// TwinCAT 3 PLC project PLC1
// ProgramVersion: 3.1.4023.0
// libraries:
//   Tc2_Utilities, * (Beckhoff Automation GmbH)
//   CmpBitmapPool, * (System)
//   Tc2_ControllerToolbox, * (Beckhoff Automation GmbH)
//   Tc2_MC2, * (Beckhoff Automation GmbH)
//   Tc2_NC, * (Beckhoff Automation GmbH)
//   Tc2_Standard, * (Beckhoff Automation GmbH)
//   Tc2_System, * (Beckhoff Automation GmbH)
//   Tc3_IoLink, * (Beckhoff Automation GmbH)
//   Tc3_Module, * (Beckhoff Automation GmbH)
//   VisuDialogs, * (System)
//   VisuSymbols,3.5.10.0,System
// project tree:
//   DUTs/ Figure.TcDUT, Mode.TcDUT
//   DUTs/CyltronicCom/ CyltronicMotionMode.TcDUT, CyltronicProcessDataInActual.TcDUT, CyltronicProcessDataInBytes.TcDUT, CyltronicProcessDataIn.TcDUT, CyltronicProcessDataOut.TcDUT, CyltronicProcessDataOutActual.TcDUT, CyltronicProcessDataOutBytes.TcDUT, CyltronicState.TcDUT
//   / GlobalTextList.TcGTLO, ImagePool.TcIPO (not stored), PLC_TASK.TcTTO, VISU_TASK.TcTTO
//   GVLs/ Config.TcGVL, GVL.TcGVL
//   POUs/ CONTROLLER.TcPOU, FBCylTronicCylinder.TcPOU, FB_FigureGenerator.TcPOU, FB_FigurePlayer.TcPOU, FB_BallTrack.TcPOU, FB_ReglerParam.TcPOU, MAIN.TcPOU, Touchpanel.TcPOU, TOUCH_SCALE.TcPOU, xy_RST_Transformation_dynamisch.TcPOU
//   POUs/Regelungstechnik/ DT1.TcPOU, eFiltertyp.TcDUT, eReglertyp.TcDUT, eSignalform.TcDUT, FB_Totband.TcPOU, Integrator.TcPOU, Logger_RET.TcPOU, P.TcPOU, PT1.TcPOU, PT2.TcPOU, PT2s.TcPOU, PTt.TcPOU, Rauschen.TcPOU, Regler.TcPOU, RET_COMMON.TcPOU, Signalgenerator.TcPOU, Strecke.TcPOU
//   POUs/Regelungstechnik/visu/ RET_VISU_DT1.TcVIS, RET_VISU_Integrator.TcVIS, RET_VISU_Kennlinie.TcVIS, RET_VISU_P.TcVIS, RET_VISU_PT1.TcVIS, RET_VISU_PT2.TcVIS, RET_VISU_PT2s.TcVIS, RET_VISU_PTt.TcVIS, RET_VISU_Regler.TcVIS, RET_VISU_Signalgenerator.TcVIS, RET_VISU_Strecke.TcVIS, TextListForCombobox_eReglertyp.TcTLO, TextListForCombobox_eSignalform.TcTLO, VISU_HELPER_Combobox_eReglertyp.TcVIS, VISU_HELPER_Combobox_eSignalform.TcVIS
//   VISUs/ Achse_R.TcVIS, Achse_S.TcVIS, Achse_T.TcVIS, FigureGeneratorDisplay.TcVIS, Home.TcVIS, FigureGenerator1.TcVIS, Debug.TcVIS, InputNumSlider_Corner.TcVIS, InputNumSlider_Radius.TcVIS, InputNumSlider_Angle.TcVIS, InputNumSlider_Time.TcVIS, Mainvisu.TcVIS, Polygon.TcVIS, FigurePlayer.TcVIS, FigureGenerator.TcVIS, FigurePlayerDisplay.TcVIS, Polygon_1.TcVIS, VisualizationManager.TcVMO (not stored), Visu_Achse.TcVIS
// real-time tasks:
//   TASK PLC_TASK: cycle T#1ms, priority 1, ADS port 350
//   TASK VISU_TASK: cycle T#200000us, priority 12, ADS port 351
// I/O:
//   DEVICE Device 2 (EtherCAT), AmsNetId 192.168.0.33.3.1
//     Klemme 1 (EK1200) [EK1200-5000 EtherCAT Netzteil (2A E-Bus)]
//       Klemme 2 (EL6224) [EL6224 (IO Link Master)]
//       Klemme 3 (EL1859) [EL1859 8K. Dig. Eingang 24V, 3ms, 8K. Dig. Ausgang 24V, 0.5A]
//       Klemme 4 (EK1110) [EK1110 EtherCAT-Verlängerung]
//     Box 14 (ABBTS Ball and Plate) [ABBTS Ball and Plate]
// variable links:
//   PLC1/PLC1 Instance <-> Device 2 (EtherCAT)/Box 14 (ABBTS Ball and Plate)
//     PLC_TASK Inputs/Touchpanel.bContactAvailable <-> Inputs/byContactAvailable
//     PLC_TASK Inputs/Touchpanel.iXadc <-> Inputs/iXraw
//     PLC_TASK Inputs/Touchpanel.iYadc <-> Inputs/iYraw
//     PLC_TASK Inputs/Touchpanel.iZadc <-> Inputs/iZraw
//     PLC_TASK Inputs/Touchpanel.rXadc <-> Inputs/rX
//     PLC_TASK Inputs/Touchpanel.rYadc <-> Inputs/rY
//     PLC_TASK Inputs/Touchpanel.rZadc <-> Inputs/rZ
//     PLC_TASK Outputs/Touchpanel.iStep <-> Outputs/iStep
//     PLC_TASK Outputs/Touchpanel.rQ_Kalman <-> Outputs/rQ_Kalman
//     PLC_TASK Outputs/Touchpanel.rR_Kalman <-> Outputs/rR_Kalman
//   PLC1/PLC1 Instance <-> Device 2 (EtherCAT)/Term 1 (EK1200)/Term 2 (EL6224)
//     PLC_TASK Inputs/MAIN.Axis_R.DataIn/CyltronicDataInByte/Byte0 <-> IO-Link Port1_in/SubIndex 001[0]
//     PLC_TASK Inputs/MAIN.Axis_R.DataIn/CyltronicDataInByte/Byte1 <-> IO-Link Port1_in/SubIndex 001[1]
//     PLC_TASK Inputs/MAIN.Axis_R.DataIn/CyltronicDataInByte/Byte10 <-> IO-Link Port1_in/SubIndex 001[10]
//     PLC_TASK Inputs/MAIN.Axis_R.DataIn/CyltronicDataInByte/Byte11 <-> IO-Link Port1_in/SubIndex 001[11]
//     PLC_TASK Inputs/MAIN.Axis_R.DataIn/CyltronicDataInByte/Byte12 <-> IO-Link Port1_in/SubIndex 001[12]
//     PLC_TASK Inputs/MAIN.Axis_R.DataIn/CyltronicDataInByte/Byte13 <-> IO-Link Port1_in/SubIndex 001[13]
//     PLC_TASK Inputs/MAIN.Axis_R.DataIn/CyltronicDataInByte/Byte2 <-> IO-Link Port1_in/SubIndex 001[2]
//     PLC_TASK Inputs/MAIN.Axis_R.DataIn/CyltronicDataInByte/Byte3 <-> IO-Link Port1_in/SubIndex 001[3]
//     PLC_TASK Inputs/MAIN.Axis_R.DataIn/CyltronicDataInByte/Byte4 <-> IO-Link Port1_in/SubIndex 001[4]
//     PLC_TASK Inputs/MAIN.Axis_R.DataIn/CyltronicDataInByte/Byte5 <-> IO-Link Port1_in/SubIndex 001[5]
//     PLC_TASK Inputs/MAIN.Axis_R.DataIn/CyltronicDataInByte/Byte6 <-> IO-Link Port1_in/SubIndex 001[6]
//     PLC_TASK Inputs/MAIN.Axis_R.DataIn/CyltronicDataInByte/Byte7 <-> IO-Link Port1_in/SubIndex 001[7]
//     PLC_TASK Inputs/MAIN.Axis_R.DataIn/CyltronicDataInByte/Byte8 <-> IO-Link Port1_in/SubIndex 001[8]
//     PLC_TASK Inputs/MAIN.Axis_R.DataIn/CyltronicDataInByte/Byte9 <-> IO-Link Port1_in/SubIndex 001[9]
//     PLC_TASK Inputs/MAIN.Axis_S.DataIn/CyltronicDataInByte/Byte0 <-> IO-Link Port2_in/SubIndex 001[0]
//     PLC_TASK Inputs/MAIN.Axis_S.DataIn/CyltronicDataInByte/Byte1 <-> IO-Link Port2_in/SubIndex 001[1]
//     PLC_TASK Inputs/MAIN.Axis_S.DataIn/CyltronicDataInByte/Byte10 <-> IO-Link Port2_in/SubIndex 001[10]
//     PLC_TASK Inputs/MAIN.Axis_S.DataIn/CyltronicDataInByte/Byte11 <-> IO-Link Port2_in/SubIndex 001[11]
//     PLC_TASK Inputs/MAIN.Axis_S.DataIn/CyltronicDataInByte/Byte12 <-> IO-Link Port2_in/SubIndex 001[12]
//     PLC_TASK Inputs/MAIN.Axis_S.DataIn/CyltronicDataInByte/Byte13 <-> IO-Link Port2_in/SubIndex 001[13]
//     PLC_TASK Inputs/MAIN.Axis_S.DataIn/CyltronicDataInByte/Byte2 <-> IO-Link Port2_in/SubIndex 001[2]
//     PLC_TASK Inputs/MAIN.Axis_S.DataIn/CyltronicDataInByte/Byte3 <-> IO-Link Port2_in/SubIndex 001[3]
//     PLC_TASK Inputs/MAIN.Axis_S.DataIn/CyltronicDataInByte/Byte4 <-> IO-Link Port2_in/SubIndex 001[4]
//     PLC_TASK Inputs/MAIN.Axis_S.DataIn/CyltronicDataInByte/Byte5 <-> IO-Link Port2_in/SubIndex 001[5]
//     PLC_TASK Inputs/MAIN.Axis_S.DataIn/CyltronicDataInByte/Byte6 <-> IO-Link Port2_in/SubIndex 001[6]
//     PLC_TASK Inputs/MAIN.Axis_S.DataIn/CyltronicDataInByte/Byte7 <-> IO-Link Port2_in/SubIndex 001[7]
//     PLC_TASK Inputs/MAIN.Axis_S.DataIn/CyltronicDataInByte/Byte8 <-> IO-Link Port2_in/SubIndex 001[8]
//     PLC_TASK Inputs/MAIN.Axis_S.DataIn/CyltronicDataInByte/Byte9 <-> IO-Link Port2_in/SubIndex 001[9]
//     PLC_TASK Inputs/MAIN.Axis_T.DataIn/CyltronicDataInByte/Byte0 <-> IO-Link Port3_in/SubIndex 001[0]
//     PLC_TASK Inputs/MAIN.Axis_T.DataIn/CyltronicDataInByte/Byte1 <-> IO-Link Port3_in/SubIndex 001[1]
//     PLC_TASK Inputs/MAIN.Axis_T.DataIn/CyltronicDataInByte/Byte10 <-> IO-Link Port3_in/SubIndex 001[10]
//     PLC_TASK Inputs/MAIN.Axis_T.DataIn/CyltronicDataInByte/Byte11 <-> IO-Link Port3_in/SubIndex 001[11]
//     PLC_TASK Inputs/MAIN.Axis_T.DataIn/CyltronicDataInByte/Byte12 <-> IO-Link Port3_in/SubIndex 001[12]
//     PLC_TASK Inputs/MAIN.Axis_T.DataIn/CyltronicDataInByte/Byte13 <-> IO-Link Port3_in/SubIndex 001[13]
//     PLC_TASK Inputs/MAIN.Axis_T.DataIn/CyltronicDataInByte/Byte2 <-> IO-Link Port3_in/SubIndex 001[2]
//     PLC_TASK Inputs/MAIN.Axis_T.DataIn/CyltronicDataInByte/Byte3 <-> IO-Link Port3_in/SubIndex 001[3]
//     PLC_TASK Inputs/MAIN.Axis_T.DataIn/CyltronicDataInByte/Byte4 <-> IO-Link Port3_in/SubIndex 001[4]
//     PLC_TASK Inputs/MAIN.Axis_T.DataIn/CyltronicDataInByte/Byte5 <-> IO-Link Port3_in/SubIndex 001[5]
//     PLC_TASK Inputs/MAIN.Axis_T.DataIn/CyltronicDataInByte/Byte6 <-> IO-Link Port3_in/SubIndex 001[6]
//     PLC_TASK Inputs/MAIN.Axis_T.DataIn/CyltronicDataInByte/Byte7 <-> IO-Link Port3_in/SubIndex 001[7]
//     PLC_TASK Inputs/MAIN.Axis_T.DataIn/CyltronicDataInByte/Byte8 <-> IO-Link Port3_in/SubIndex 001[8]
//     PLC_TASK Inputs/MAIN.Axis_T.DataIn/CyltronicDataInByte/Byte9 <-> IO-Link Port3_in/SubIndex 001[9]
//     PLC_TASK Outputs/MAIN.Axis_R.DataOut/CyltronicDataOutByte/Byte0 <-> IO-Link Port1_out/SubIndex 001[0]
//     PLC_TASK Outputs/MAIN.Axis_R.DataOut/CyltronicDataOutByte/Byte1 <-> IO-Link Port1_out/SubIndex 001[1]
//     PLC_TASK Outputs/MAIN.Axis_R.DataOut/CyltronicDataOutByte/Byte2 <-> IO-Link Port1_out/SubIndex 001[2]
//     PLC_TASK Outputs/MAIN.Axis_R.DataOut/CyltronicDataOutByte/Byte3 <-> IO-Link Port1_out/SubIndex 001[3]
//     PLC_TASK Outputs/MAIN.Axis_R.DataOut/CyltronicDataOutByte/Byte4 <-> IO-Link Port1_out/SubIndex 001[4]
//     PLC_TASK Outputs/MAIN.Axis_R.DataOut/CyltronicDataOutByte/Byte5 <-> IO-Link Port1_out/SubIndex 001[5]
//     PLC_TASK Outputs/MAIN.Axis_R.DataOut/CyltronicDataOutByte/Byte6 <-> IO-Link Port1_out/SubIndex 001[6]
//     PLC_TASK Outputs/MAIN.Axis_R.DataOut/CyltronicDataOutByte/Byte7 <-> IO-Link Port1_out/SubIndex 001[7]
//     PLC_TASK Outputs/MAIN.Axis_S.DataOut/CyltronicDataOutByte/Byte0 <-> IO-Link Port2_out/SubIndex 001[0]
//     PLC_TASK Outputs/MAIN.Axis_S.DataOut/CyltronicDataOutByte/Byte1 <-> IO-Link Port2_out/SubIndex 001[1]
//     PLC_TASK Outputs/MAIN.Axis_S.DataOut/CyltronicDataOutByte/Byte2 <-> IO-Link Port2_out/SubIndex 001[2]
//     PLC_TASK Outputs/MAIN.Axis_S.DataOut/CyltronicDataOutByte/Byte3 <-> IO-Link Port2_out/SubIndex 001[3]
//     PLC_TASK Outputs/MAIN.Axis_S.DataOut/CyltronicDataOutByte/Byte4 <-> IO-Link Port2_out/SubIndex 001[4]
//     PLC_TASK Outputs/MAIN.Axis_S.DataOut/CyltronicDataOutByte/Byte5 <-> IO-Link Port2_out/SubIndex 001[5]
//     PLC_TASK Outputs/MAIN.Axis_S.DataOut/CyltronicDataOutByte/Byte6 <-> IO-Link Port2_out/SubIndex 001[6]
//     PLC_TASK Outputs/MAIN.Axis_S.DataOut/CyltronicDataOutByte/Byte7 <-> IO-Link Port2_out/SubIndex 001[7]
//     PLC_TASK Outputs/MAIN.Axis_T.DataOut/CyltronicDataOutByte/Byte0 <-> IO-Link Port3_out/SubIndex 001[0]
//     PLC_TASK Outputs/MAIN.Axis_T.DataOut/CyltronicDataOutByte/Byte1 <-> IO-Link Port3_out/SubIndex 001[1]
//     PLC_TASK Outputs/MAIN.Axis_T.DataOut/CyltronicDataOutByte/Byte2 <-> IO-Link Port3_out/SubIndex 001[2]
//     PLC_TASK Outputs/MAIN.Axis_T.DataOut/CyltronicDataOutByte/Byte3 <-> IO-Link Port3_out/SubIndex 001[3]
//     PLC_TASK Outputs/MAIN.Axis_T.DataOut/CyltronicDataOutByte/Byte4 <-> IO-Link Port3_out/SubIndex 001[4]
//     PLC_TASK Outputs/MAIN.Axis_T.DataOut/CyltronicDataOutByte/Byte5 <-> IO-Link Port3_out/SubIndex 001[5]
//     PLC_TASK Outputs/MAIN.Axis_T.DataOut/CyltronicDataOutByte/Byte6 <-> IO-Link Port3_out/SubIndex 001[6]
//     PLC_TASK Outputs/MAIN.Axis_T.DataOut/CyltronicDataOutByte/Byte7 <-> IO-Link Port3_out/SubIndex 001[7]
//   PLC1/PLC1 Instance <-> Device 2 (EtherCAT)/Term 1 (EK1200)/Term 3 (EL1859)
//     PLC_TASK Inputs/GVL.NOTAUS <-> Channel 3/Input
//     PLC_TASK Inputs/GVL.Netzgeraet48VOK <-> Channel 2/Input
//     PLC_TASK Inputs/GVL.V48DC_Ein <-> Channel 1/Input
//     PLC_TASK Outputs/GVL.V48Einbefehl <-> Channel 9/Output

CONFIGURATION PLC1
    RESOURCE PLC ON TwinCAT3
        TASK PLC_TASK(INTERVAL := T#1ms, PRIORITY := 1);
        TASK VISU_TASK(INTERVAL := T#200000us, PRIORITY := 12);
        PROGRAM MAIN WITH PLC_TASK : MAIN;
        PROGRAM VisuElems_Visu_Prg WITH VISU_TASK : VisuElems.Visu_Prg;
    END_RESOURCE
END_CONFIGURATION

// ---- DUTs/Figure.TcDUT
TYPE Figure :
STRUCT
	length : UDINT := 0;
    X : ARRAY[0..999999] OF REAL := [100000(0)];
    Y : ARRAY[0..999999] OF REAL := [100000(0)];
	Visu : ARRAY[0..999] OF VisuElems.VisuStructPoint;
	VisuLenght : INT := 0;
	pVisu : POINTER TO ARRAY[0..999] OF VisuElems.VisuStructPoint;
END_STRUCT
END_TYPE

// ---- DUTs/Mode.TcDUT
{attribute 'qualified_only'}
{attribute 'strict'}
TYPE Mode :
(
	Off,
	Position,
	Homing,
	BallundPlate,
	Sinus,
	Tilt
);
END_TYPE

// ---- DUTs/CyltronicCom/CyltronicMotionMode.TcDUT
{attribute 'qualified_only'}
{attribute 'strict'}
TYPE CyltronicMotionMode :
(
	Off 		:= 0,
	DIO 		:= 1,
	Teach 		:= 2,
	MoveOut 	:= 3,
	MoveIn 		:= 4,
	FreePos 	:= 5,
	FreePosPro 	:= 6,
	HomeDirect 	:= 7,
	Reset		:= 255
)USINT;
END_TYPE

// ---- DUTs/CyltronicCom/CyltronicProcessDataInActual.TcDUT
{attribute 'pack_mode' := '0'}
TYPE CyltronicProcessDataInActual :
STRUCT
	State 							: CyltronicState;
	Ready 							: BIT;
	Homed 							: BIT;
	LimitSwitchOut 					: BIT;
	LimitSwitchIn 					: BIT;
	MotionModeActive 				: BIT;
	MotionCommandCompleted 			: BIT;
	WarningActive 					: BIT;
	TrackingErrorToleranceExceeded 	: BIT;
	ActualPosition 					: REAL;
	ActualSpeed 					: REAL;
	ActualForce 					: REAL;
END_STRUCT
END_TYPE

// ---- DUTs/CyltronicCom/CyltronicProcessDataInBytes.TcDUT
{attribute 'pack_mode' := '0'}
TYPE CyltronicProcessDataInBytes :
STRUCT
	Byte0  : BYTE;
	Byte1  : BYTE;
	Byte5  : BYTE;
	Byte4  : BYTE;
	Byte3  : BYTE;
	Byte2  : BYTE;
	Byte9  : BYTE;
	Byte8  : BYTE;
	Byte7  : BYTE;
	Byte6  : BYTE;
	Byte13 : BYTE;
	Byte12 : BYTE;
	Byte11 : BYTE;
	Byte10 : BYTE;
END_STRUCT
END_TYPE

// ---- DUTs/CyltronicCom/CyltronicProcessDataIn.TcDUT
TYPE CyltronicProcessDataIn :
UNION
	CyltronicDataInAct  : CyltronicProcessDataInActual;
	CyltronicDataInByte : CyltronicProcessDataInBytes;
END_UNION
END_TYPE

// ---- DUTs/CyltronicCom/CyltronicProcessDataOut.TcDUT
TYPE CyltronicProcessDataOut :
UNION
	CyltronicDataOutAct  : CyltronicProcessDataOutActual;
	CyltronicDataOutByte : CyltronicProcessDataOutBytes;
END_UNION
END_TYPE

// ---- DUTs/CyltronicCom/CyltronicProcessDataOutActual.TcDUT
{attribute 'pack_mode' := '0'}
TYPE CyltronicProcessDataOutActual :
STRUCT
	MotionMode 			 : CyltronicMotionMode;
	TargetPosition 		 : REAL;
	SpeedOverride 		 : USINT;
	ForceOverride 		 : USINT;
	AccelerationOverride : USINT;
END_STRUCT
END_TYPE

// ---- DUTs/CyltronicCom/CyltronicProcessDataOutBytes.TcDUT
{attribute 'pack_mode' := '0'}
TYPE CyltronicProcessDataOutBytes :
STRUCT
	Byte0  : BYTE;
	Byte4  : BYTE;
	Byte3  : BYTE;
	Byte2  : BYTE;
	Byte1  : BYTE;
	Byte5  : BYTE;
	Byte6  : BYTE;
	Byte7  : BYTE;
END_STRUCT
END_TYPE

// ---- DUTs/CyltronicCom/CyltronicState.TcDUT
{attribute 'qualified_only'}
{attribute 'strict'}
TYPE CyltronicState :
(
	Idle 	:= 0,
	Ready 	:= 1,
	Active 	:= 2,
	Error 	:= 3,
	Teach 	:= 4
)USINT;
END_TYPE

// ---- POUs/Regelungstechnik/eFiltertyp.TcDUT
TYPE eFiltertyp :
(
	NONE_ := 1,
	TIEFPASS := 2,
	HOCHPASS := 3
);
END_TYPE

// ---- POUs/Regelungstechnik/eReglertyp.TcDUT
TYPE eReglertyp :
(
	P := 1,
	I := 2,
	PI := 3,
	PDT1 := 4,
	PIDT1 := 5
);
END_TYPE

// ---- POUs/Regelungstechnik/eSignalform.TcDUT
TYPE eSignalform :
(
	OFF := 1,
	OFFSET := 2,
	RECHTECK := 3,
	DREIECK := 4,
	SINUS := 5
);
END_TYPE

// ---- GVLs/Config.TcGVL
{attribute 'Tc2GvlVarNames'}
VAR_GLOBAL
	IO_Link_AMS AT %I* 	: T_AmsNetId := '192.168.0.33.2.3';
	ADDRCyl1			: E_IolPort := 1;
	ADDRCyl2			: E_IolPort := 2;
	ADDRCyl3			: E_IolPort := 3;
	MaxSpeed_ADR 		: BYTE := 16#42;
	MaxForce_ADR 		: BYTE := 16#54;
	MaxACC_ADR 			: BYTE := 16#44;
	MaxDEC_ADR 			: BYTE := 16#45;
	MaxTrackingErr_ADR 	: BYTE := 16#46;

	MaxVelo 			: REAL := 300/2.55;			//max Speed in Freepositioning Mode set in Cylinder[mm/s]
	MaxForce 			: REAL := 800/2.55;			//max Force set in Cylinder [N]
	MaxACC 				: REAL := 15/2.55;			//max Acceleration (and Deceleration) set in Cylinder [mm/s^2]
	MaxTrackingErr 		: REAL := 5;				//max Tracking Error (Schleppfehler) [mm]
	MaxTravel			: REAL := 200;				//max Travel of Axis [mm]
END_VAR

// ---- GVLs/GVL.TcGVL
{attribute 'qualified_only'}
VAR_GLOBAL
	//Inputs von Visu an System
	Einbefehl: BOOL;
	Automatik:BOOL;
	Homing:BOOL;
	Grundposition:BOoL;
	Down, Up:BOOL;
	Eingabe_Grundposition:REAL:=0;
	Eingabe_Sollposition:REAL:=100;
	StepSize:INT:=1;
	BndP:BOOL;
	Sinus:BOOL;
	YAchseUp:BOOL;
	YAchseDown:BOOL;
	XAchseUp:BOOL;
	XAchseDown:BOOL;
	Tilt:BOOL;
	reset:BOOL;
	
	//Allgemeine Outputs an Visu vom System
	Warnung_Steigungswinkel:BOOL:=FALSE;
	
	//Outputs von Allgemein ans System
	eingabesperre:BOOL;
	Achsenkontrolle:BOOL;
	Position_Aktiv:BOOL;
	Sinus_Aktiv:BOOL;
	BNP_Aktiv:BOOL;
	
	//Inputs SPS
	V48DC_Ein AT %I* :BOOL;
	Netzgeraet48VOK AT %I* :BOOL;
	NOTAUS AT %I* :BOOL;
	
	
	//Outputs SPS
	V48Einbefehl AT %Q* :BOOL;
	
	rTasktime : REAL := 0.001; // Tasktime [s]
END_VAR

// ---- POUs/MAIN.TcPOU
PROGRAM MAIN
VAR_INPUT
	Axis_S				: FBCylTronicCylinder;
	Axis_T				: FBCyltronicCylinder;
	Axis_R				: FBCyltronicCylinder;
	rSetPos_R			: REAL := 0;
	rSetPos_S			: REAL := 0;
	rSetPos_T			: REAL := 0;
END_VAR

VAR
	Sinus				: FB_CTRL_SIGNAL_GENERATOR;
	SinusParams			: ST_CTRL_SIGNAL_GENERATOR_PARAMS;
	SinusMode			: E_CTRL_MODE := E_CTRL_MODE.eCTRL_MODE_ACTIVE;
	rXBallPos			: REAL; //Ball Position X Axis in mm
	rYBallPos			: REAL; //Ball Position Y Axis in mm
	rMaxTouchPos		: REAL := 363 / 2;
	rSetVelo			: REAL := 300;
	rSetAcc				: REAL := 2;
	rSetForce			: REAL := 800;
	Modus				: Mode;
	trigDown, trigUp	: R_TRIG;
	bDOWN, bUp			: BOOL;
	bBallOnPlate		: BOOL;
	bBallonPlateButton	: BOOL := FALSE;
	FB_FigureGenerator	: FB_FigureGenerator;
	FB_BallTrack		: FB_BallTrack;
END_VAR

Axis_R(stAxisName:='Achse 1');
Axis_S(stAxisName:='Achse 2');
Axis_T(stAxisName:='Achse 3');
Touchpanel();
AC_ModeSelection();
AC_TouchPos();
CONTROLLER();
FB_FigureGenerator();
FB_BallTrack();

ACTION AC_ModeSelection:

//Ausschaltbedingungen (Prio 1)
IF NOT gvl.Einbefehl OR NOT gvl.NOTAUS THEN
	Axis_R.bEnable := FALSE;
	Axis_S.bEnable := FALSE;
	Axis_T.bEnable := FALSE;
	Modus := Mode.Off;
	GVL.V48Einbefehl := FALSE;
END_IF

IF NOT GVL.NOTAUS THEN
	GVL.Einbefehl := FALSE;
END_IF

//Resetbefehl
IF gvl.reset THEN
	Axis_R.bReset := TRUE;
	Axis_S.bReset := TRUE;
	Axis_T.bReset := TRUE;
	Modus := Mode.Off;
END_IF

Axis_R.rSetForce	:= rSetForce;
Axis_S.rSetForce	:= rSetForce;
Axis_T.rSetForce	:= rSetForce;
Axis_R.rSetAcc		:= rSetAcc;
Axis_S.rSetAcc		:= rSetAcc;
Axis_T.rSetAcc		:= rSetAcc;
Axis_R.rSetVelo		:= rSetVelo;
Axis_S.rSetVelo		:= rSetVelo;
Axis_T.rSetVelo		:= rSetVelo;
Axis_R.bHoming 		:= FALSE;
Axis_S.bHoming 		:= FALSE;
Axis_T.bHoming 		:= FALSE;

IF (NOT Axis_R.Ready OR NOT Axis_S.Ready OR NOT Axis_T.Ready) AND gvl.Einbefehl AND gvl.NOTAUS THEN
	GVL.V48Einbefehl := TRUE;
	Modus := Mode.Homing;
ELSIF GVL.Grundposition THEN
	Modus := Mode.Position;
ELSIF gvl.BndP THEN
	Modus:=Mode.BallundPlate;
ELSIF gvl.Sinus THEN
	Modus:=Mode.Sinus;
ELSIF GVL.Tilt THEN
	Modus:=Mode.Tilt;
ELSIF gvl.Homing THEN
	Modus:=Mode.Homing;
END_IF

GVL.Sinus_Aktiv := FALSE;
GVL.BNP_Aktiv	:= FALSE;
IF Modus <> Mode.BallundPlate THEN
	bBallOnPlateButton := FALSE;
	bBallOnPlate := FALSE;
END_IF

CASE Modus OF
	Mode.Off:
		;
		
	Mode.Homing:
		Axis_R.bEnable := TRUE;
		Axis_S.bEnable := TRUE;
		Axis_T.bEnable := TRUE;
		Axis_R.bHoming := TRUE;
		Axis_S.bHoming := TRUE;
		Axis_T.bHoming := TRUE;
		gvl.eingabesperre:=TRUE;
		
	Mode.Position:
		IF gvl.Automatik THEN
			rSetPos_R := rSetPos_S := rSetPos_T	:= gvl.Eingabe_Sollposition;
		END_IF
	
	Mode.Tilt:
		;
	
	Mode.Sinus:
		SinusParams.eSignalType := E_CTRL_SIGNAL_TYPE.eCTRL_SINUS;
		SinusParams.fAmplitude := (MaxTravel - 2 ) / 2;
		SinusParams.fOffset := MaxTravel / 2;
		SinusParams.tCtrlCycleTime := T#2MS;
		SinusParams.tCylceDuration := T#2S;
		SinusParams.tTaskCycleTime := T#2MS;
		Sinus(stParams := SinusParams);
		Sinus.eMode := SinusMode;
		rSetPos_R := rSetPos_S := rSetPos_T := LREAL_TO_REAL(Sinus.fOut);
	
	Mode.BallundPlate:
		bBallOnPlate := bBallOnPlateButton;
	
		;
END_CASE
Axis_R.rSetPos	:= rSetPos_R;
Axis_S.rSetPos	:= rSetPos_S;
Axis_T.rSetPos	:= rSetPos_T;
END_ACTION

ACTION AC_TouchPos:
IF CONTROLLER.bReAktiv THEN
	rXBallPos := Touchpanel.touch_scale_x.rX_mm;
	rYBallPos := Touchpanel.touch_scale_y.rX_mm;
ELSE
	rXBallPos := -180;
	rYBallPos := -142;
END_IF
END_ACTION

END_PROGRAM

// ---- POUs/FBCylTronicCylinder.TcPOU
FUNCTION_BLOCK FBCylTronicCylinder
VAR_INPUT
	DataIn AT %I*	: CyltronicProcessDataIn;
	rSetPos			: REAL;
	rSetVelo		: REAL;
	rSetForce		: REAL;
	rSetAcc			: REAL;
	bEnable			: BOOL;
	bReset			: BOOL;
	bHoming			: BOOL;
	stAxisName		: STRING;
END_VAR
VAR_OUTPUT
	DataOut AT %Q* : CyltronicProcessDataOut;
END_VAR
VAR
	bManual, bUp, bDown				: BOOL;
	UpTRIG, DownTRIG				: R_TRIG;
	iPosOffset						: INT	:= 0;
	ActualForce						: REAL;
	ActualPosition					: REAL;
	ActualSpeed						: REAL;
	LimitSwitchIn					: BOOL;
	LimitSwitchOut					: BOOL;
	MotionCommandCompleted			: BOOL;
	MotionModeActive				: BOOL;
	Ready							: BOOL;
	WarningActive					: BOOL;
	TrackingErrorToleranceExceeded	: BOOL;
	CylState						: REAL;
	Position_Aktiv					: BOOL;
	Sinus_Aktiv						: BOOL;
	BNP_Aktiv						: BOOL;
	TonError						: TON;
END_VAR

UpTRIG(CLK:=bUp);
DownTRIG(CLK:=bDown);
TonError(IN := bHoming, PT := T#20MS);

IF bReset THEN
	DataOut.CyltronicDataOutAct.MotionMode			:= CyltronicMotionMode.Reset;
	bReset 											:= FALSE;
ELSIF NOT bEnable THEN
	DataOut.CyltronicDataOutAct.MotionMode 			:= CyltronicMotionMode.Off;
	DataOut.CyltronicDataOutAct.TargetPosition 		:= DataIn.CyltronicDataInAct.ActualPosition;
	bManual 										:= FALSE;
ELSIF bHoming THEN
	IF DataIn.CyltronicDataInAct.State = CyltronicState.Error AND NOT TonError.Q THEN
		DataOut.CyltronicDataOutAct.MotionMode			:= CyltronicMotionMode.Reset;
		DataOut.CyltronicDataOutAct.TargetPosition		:= DataIn.CyltronicDataInAct.ActualPosition;
	ELSE
		DataOut.CyltronicDataOutAct.MotionMode			:= CyltronicMotionMode.MoveIn;
	END_IF
ELSIF NOT bManual THEN
	DataOut.CyltronicDataOutAct.TargetPosition		:= LIMIT(0,rSetPos,MaxTravel);
	DataOut.CyltronicDataOutAct.MotionMode			:= CyltronicMotionMode.FreePosPro;
ELSE
	IF UpTrig.Q AND iPosOffset < MaxTravel THEN
		iPosOffset := iPosOffset + GVL.StepSize;
	ELSIF DownTrig.Q AND iPosOffset > - MaxTravel THEN
		iPosOffset := iPosOffset - GVL.StepSize;
	END_IF
	DataOut.CyltronicDataOutAct.TargetPosition		:= LIMIT(0,rSetPos + iPosOffset,MaxTravel);
	DataOut.CyltronicDataOutAct.MotionMode			:= CyltronicMotionMode.FreePosPro;
	//iPosOffset := 0;
END_IF

//Outputs
DataOut.CyltronicDataOutAct.AccelerationOverride 	:= LIMIT(1, REAL_TO_USINT(rSetAcc / MaxACC * 100), 255);
DataOut.CyltronicDataOutAct.ForceOverride 			:= LIMIT(1, REAL_TO_USINT(rSetForce / MaxForce * 100), 255);
DataOut.CyltronicDataOutAct.SpeedOverride 			:= LIMIT(1, REAL_TO_USINT(rSetVelo / MaxVelo * 100), 255);

ActualForce											:= DataIn.CyltronicDataInAct.ActualForce;
ActualPosition										:= DataIn.CyltronicDataInAct.ActualPosition;
ActualSpeed											:= DataIn.CyltronicDataInAct.ActualSpeed;
LimitSwitchIn										:= DataIn.CyltronicDataInAct.LimitSwitchIn;
LimitSwitchOut										:= DataIn.CyltronicDataInAct.LimitSwitchOut;
MotionCommandCompleted								:= DataIn.CyltronicDataInAct.MotionCommandCompleted;
MotionModeActive									:= DataIn.CyltronicDataInAct.MotionModeActive;
Ready												:= DataIn.CyltronicDataInAct.Ready;
WarningActive										:= DataIn.CyltronicDataInAct.WarningActive;
TrackingErrorToleranceExceeded						:= DataIn.CyltronicDataInAct.TrackingErrorToleranceExceeded;
CylState											:= DataIn.CyltronicDataInAct.State;

END_FUNCTION_BLOCK

// ---- POUs/FB_FigureGenerator.TcPOU
FUNCTION_BLOCK FB_FigureGenerator
VAR_INPUT
	bGenerate		: BOOL; //generate Figure
	bStar			: BOOL; // generate Star if True
	bClockwise		: BOOL; // clockwise Figure
	bContinus		: BOOL; // Figure continus or Point to Point?
	nCornerCountInp	: UINT := 5; //how many corners to generate
	rRadius1		: REAL := 50;  //Radius from center to a corner
	rRadius2		: REAL := 10;  //Radius from center to a corner
	rAngleOffset	: REAL := 0; //Offset of the Figure angle
	rFigureTime		: REAL := 5; //Time for the whole figure [S]
END_VAR
VAR_OUTPUT
	pFigure : POINTER TO Figure;
END_VAR
VAR 
	bStarIntern : BOOL;
	rRadius : REAL;
	rRadius_next : REAL;
	nCornerCount : UINT;
	PI		: REAL := 4 * ATAN(1);
	angle : REAL;
	x_corner : REAL;
	y_corner  : REAL;
	angle_next : REAL;
	x_corner_next  : REAL;
	y_corner_next  : REAL;
	edge_length : REAL;
	Step : REAL := 0;
	counter : UINT := 0;
	counter1 : UDINT := 0;
	counter2 : UDINT := 0;
	Figure : Figure;
	rEdgeTime : REAL;
	points_on_edge : UDINT;
	adjusted_a : REAL;
	counterOffset : REAL;
	counterOffser_next : REAL;
	a : REAL;
	rAngleOffsetRad	: REAL;
	nDir : INT := 1;
	Visu : ARRAY[0..999] OF VisuElems.VisuStructPoint;
	VisuLenght : INT := 0;
	pVisu : POINTER TO ARRAY[0..999] OF VisuElems.VisuStructPoint;
	bStarOld			: BOOL; 
	bClockwiseOld		: BOOL; 
	nCornerCountInpOld	: UINT;
	rRadius1Old			: REAL;
	rRadius2Old			: REAL;
	rAngleOffsetOld		: REAL;
	sRadius1			: STRING := 'Radius 1';
	sRadius2			: STRING := 'Radius 2';
END_VAR

 //Parameters
(*a = 5  // Distance between points
n = 10 // Number of corners
r = 80  // Radius from center to a corner*)
pFigure := ADR(Figure);
rFigureTime := LIMIT(0.01,rFigureTime, 100);
nCornerCountInp := LIMIT(3,nCornerCountInp, 100);
rEdgeTime := rFigureTime / nCornerCount *1000;
counter2 := 0;

IF bGenerate THEN
	FOR counter := 0 TO nCornerCount-1 BY 1 DO
		IF bStarIntern AND counter MOD 2 = 0 THEN
			rRadius := rRadius1;
			rRadius_next := rRadius2;
		ELSIF bStarIntern AND counter MOD 2 <> 0 THEN
			rRadius := rRadius2;
			rRadius_next := rRadius1;
		ELSE
			rRadius := rRadius1;
			rRadius_next := rRadius1;
		END_IF
		// Calculate corner coordinates
		angle := 2 * PI * (UINT_TO_REAL(counter) / UINT_TO_REAL(nCornerCount) * INT_TO_REAL(nDir) + rAngleOffsetRad) ;
		x_corner := rRadius * COS(angle);
		y_corner := rRadius * SIN(angle);
	
		// Calculate next corner coordinates
		angle_next := 2 * PI * (UINT_TO_REAL(counter + 1) / UINT_TO_REAL(nCornerCount) * INT_TO_REAL(nDir) + rAngleOffsetRad) ;
		x_corner_next := rRadius_next * COS(angle_next);
		y_corner_next := rRadius_next * SIN(angle_next);
	
		// Calculate the distance between corners (edge length)
		edge_length := LREAL_TO_REAL(SQRT(EXPT(x_corner_next - x_corner,2) + EXPT(y_corner_next - y_corner,2)));
	
		// Adjust a for this edge to fit perfectly
		a:= edge_length / rEdgeTime;
		points_on_edge := REAL_TO_UINT(edge_length / a); 
		adjusted_a := edge_length / UDINT_TO_REAL(points_on_edge);   
	
		// Generate points on this edge
		Figure.Visu[counter].iX := REAL_TO_INT((x_corner)+ 392/2)*3;
		Figure.Visu[counter].iY := REAL_TO_INT((-y_corner)+ 318/2)*3;
		FOR counter1 := 0 TO points_on_edge-1 DO
			IF bContinus THEN
				Figure.X[counter2] := x_corner + UDINT_TO_REAL(counter1) * adjusted_a * (x_corner_next - x_corner) / edge_length;
				Figure.Y[counter2] := y_corner + UDINT_TO_REAL(counter1) * adjusted_a * (y_corner_next - y_corner) / edge_length;
			ELSE
				Figure.X[counter2] := x_corner;
				Figure.Y[counter2] := y_corner;
			END_IF
			counter2 := counter2 +1;
		END_FOR
 	END_FOR
	Figure.Visu[counter].iX := REAL_TO_INT((x_corner_next)+ 392/2)*3;
	Figure.Visu[counter].iY := REAL_TO_INT((-y_corner_next)+ 318/2)*3;
	Figure.VisuLenght := UINT_TO_INT(nCornerCount + 1);
 	Figure.length := counter2;
	Figure.pVisu := ADR(Figure.Visu);
	bGenerate := FALSE;
ELSE
	IF bClockwise THEN
		nDir := -1;
	ELSE
		nDir := 1;
	END_IF
	IF bStar THEN
		nCornerCount := 2 * nCornercountInp;
		bStarIntern := TRUE;
	ELSE
		nCornerCount := nCornercountInp;
		bStarIntern := FALSE;
	END_IF
	rAngleOffsetRad := rAngleOffset / 360;
	IF bStar			<>	bStarOld			OR
		nCornerCountInp	<>	nCornerCountInpOld	OR
		bClockwise		<>	bClockwiseOld		OR
		rRadius1		<>	rRadius1Old			OR
		rRadius2		<>	rRadius2Old			OR
		rAngleOffset	<>	rAngleOffsetOld		THEN;
		bStarOld			:= bStar;
		bClockwiseOld		:= bClockwise;
		nCornerCountInpOld	:= nCornerCountInp;
		rRadius1Old			:= rRadius1;
		rRadius2Old			:= rRadius2;
		rAngleOffsetOld		:= rAngleOffset;
		FOR counter := 0 TO nCornerCount-1 BY 1 DO
			IF bStarIntern AND counter MOD 2 = 0 THEN
				rRadius := rRadius1;
				rRadius_next := rRadius2;
			ELSIF bStarIntern AND counter MOD 2 <> 0 THEN
				rRadius := rRadius2;
				rRadius_next := rRadius1;
			ELSE
				rRadius := rRadius1;
				rRadius_next := rRadius1;
			END_IF
			// Calculate corner coordinates
			angle := 2 * PI * (UINT_TO_REAL(counter) / UINT_TO_REAL(nCornerCount) * INT_TO_REAL(nDir) + rAngleOffsetRad) ;
			x_corner := rRadius * COS(angle);
			y_corner := rRadius * SIN(angle);
		
			// Calculate next corner coordinates
			angle_next := 2 * PI * (UINT_TO_REAL(counter + 1) / UINT_TO_REAL(nCornerCount) * INT_TO_REAL(nDir) + rAngleOffsetRad);
			x_corner_next := rRadius_next * COS(angle_next);
			y_corner_next := rRadius_next * SIN(angle_next);  
		
			// Generate points on this edge
			Visu[counter].iX := REAL_TO_INT((x_corner)+ 392/2)*3;
			Visu[counter].iY := REAL_TO_INT((-y_corner)+ 318/2)*3;
		END_FOR
		Visu[counter].iX := REAL_TO_INT((x_corner_next)+ 392/2)*3;
		Visu[counter].iY := REAL_TO_INT((-y_corner_next)+ 318/2)*3;
		VisuLenght := UINT_TO_INT(nCornerCount + 1);
		pVisu := ADR(Visu);
		bGenerate := FALSE;
	END_IF	
END_IF

END_FUNCTION_BLOCK

// ---- POUs/FB_BallTrack.TcPOU
FUNCTION_BLOCK FB_BallTrack
VAR	
	Visu : ARRAY[0..999] OF VisuElems.VisuStructPoint;
	VisuLenght : INT := 200;
	pVisu : POINTER TO ARRAY[0..999] OF VisuElems.VisuStructPoint;
	counter: INT;
	counter1: INT := 0;
END_VAR

IF counter1 >= 100 THEN
	FOR counter := 0 TO VisuLenght-1 DO
		Visu[counter].iX := Visu[counter+1].iX;
		Visu[counter].iY := Visu[counter+1].iY;	
	END_FOR
	Visu[counter].iX := REAL_TO_INT((CONTROLLER.rX_x)+ 392/2)*3;
	Visu[counter].iY := REAL_TO_INT((-CONTROLLER.rX_y)+ 318/2)*3;
	counter1 := 0;
END_IF
counter1 := counter1 + 1;
pVisu := ADR(Visu);

END_FUNCTION_BLOCK

// ---- POUs/CONTROLLER.TcPOU
PROGRAM CONTROLLER
VAR
	/// Freigabe Regler
	bReAktiv: BOOL := FALSE;
	/// Freigabe AWU Regler
	bAwuAktiv: BOOL := TRUE;
	/// Logger
	bLoggerRunning: BOOL := FALSE;
	fbLogger: Logger_RET;
	bFilterAktiv: BOOL;
	xy_RST_Transformation_dynamisch_0: xy_RST_Transformation_dynamisch;
	rW_x: REAL;
	rW_y: REAL;
	rX_x: REAL;
	rX_y: REAL;
	rY_x: REAL;
	rY_y: REAL;
	rY_R: REAL;
	rY_S: REAL;
	rY_T: REAL;
	bEnable_Limitierung_rY_RST: BOOL := TRUE;
	rUL_rY_RST: REAL := 199;
	rLL_rY_RST: REAL := 1;
	rE_x: REAL;
	rX_y_1: REAL;
	rX_x_1: REAL;
	
	fbFilter_X_y: PT2 := (fK := 1.0, fT1 := 0.05, fT2 := 0.05);
	fbFilter_X_x: PT2 := (fK := 1.0, fT1 := 0.05, fT2 := 0.05);
	fbSignalgeno_W_y: Signalgenerator := (eTyp := eSignalform.OFFSET, fOffset := 0.0, fAmplitude := 10.0, fFrequenz := 0.25);
	fbSignalgeno_W_x: Signalgenerator := (eTyp := eSignalform.OFFSET, fOffset := 0.0, fAmplitude := 10.0, fFrequenz := 0.25);
	fbSignalgeno_Y_x: Signalgenerator := (eTyp := eSignalform.OFFSET, fOffset := 10.0, fAmplitude := 10.0, fFrequenz := 0.25);
	fbSignalgeno_Y_y: Signalgenerator := (eTyp := eSignalform.OFFSET, fOffset := 10.0, fAmplitude := 10.0, fFrequenz := 0.25);
	fbRegler_x: Regler;
	fbRegler_y: Regler;
	
	
	rE_y: REAL;
	rAxisOffset: REAL := 100;
	// Zusätzlicher Filter auf Stellgrösse RST
	y_r_filter: PT1 := (fK := 1, fT := 0.05);
	y_s_filter: PT1 := (fK := 1, fT := 0.05);
	y_t_filter: PT1 := (fK := 1, fT := 0.05);
	ry_rst_filter: REAL := 0.0;  // Filterzeitkonstante PT1
	rContactTime: TIME := T#0.5s;
	flim_max : REAL :=30;
	flim_min : REAL :=-30;
	PT2_E_y: PT2;
	FB_Totband_x: FB_Totband;
	FB_Totband_y: FB_Totband;
	FB_ReglerParam_x: FB_ReglerParam;
	FB_ReglerParam_y: FB_ReglerParam;
	ControllerNum : UINT := 0;
	TON_Touch: TON;
	TOF_Touch: TOF;
	rX_r: REAL;
	FB_FigurePlayer_0: FB_FigurePlayer;
END_VAR
VAR // added by the converter: edge detectors and wires of the graphical bodies
    _w1, _w2 : BOOL;
    _w3, _w4, _w5, _w10, _w11, _w12, _w13, _w15, _w16, _w18 : ANY;
    _w6, _w7, _w8, _w9, _w14, _w17 : REAL;
END_VAR

_w1 := MAIN.Modus = Mode.BallundPlate;
bReAktiv := _w2;
FB_Totband_y(rTotband := FB_ReglerParam_y.rTotband, rPos := _w3); // FB_Totband
FB_ReglerParam_x(ControllerNum := ControllerNum); // FB_ReglerParam
MAIN.rSetPos_T := _w4;
_w5 := fbFilter_X_x.fY / MAIN.rMaxTouchPos;
TON_Touch(IN := TOF_Touch.Q, PT := rContactTime); // TON
_w6 := BOOL_TO_REAL(Touchpanel.bContactAvailable);
TOF_Touch(IN := Touchpanel.bContactAvailable, PT := rContactTime); // TOF
_w7 := _w6 * 100;
FB_FigurePlayer_0(
    pFigure := MAIN.FB_FigureGenerator.pFigure,
    rW_xIn := fbSignalgeno_W_x.fY,
    rW_yIn := fbSignalgeno_W_y.fY); // FB_FigurePlayer
_w2 := TON_Touch.Q AND _w1;
// Vorgabe im
// gesteuerten Betrieb
fbSignalgeno_Y_x(); // Signalgenerator
rX_y_1 := _w8;
fbSignalgeno_W_x(); // Signalgenerator
// Regelglied
rW_x := FB_FigurePlayer_0.rW_x;
fbFilter_X_x(fX := MAIN.rXBallPos); // PT2
_w9 := rW_x - rX_x;
// Sollwert
rE_x := _w9;
fbRegler_x(
    fE := FB_Totband_x.rPosFilt,
    eTyp := FB_ReglerParam_x.Reglertyp,
    bReset := NOT bReAktiv,
    fKr := FB_ReglerParam_x.KP,
    fTn := FB_ReglerParam_x.Ti,
    fTv := FB_ReglerParam_x.Td,
    fTvz := FB_ReglerParam_x.Tvz,
    bEnable_AWU := bAwuAktiv,
    fYlim_max := flim_max,
    fYlim_min := flim_min); // Regler
rY_x := SEL(bReAktiv, fbSignalgeno_Y_x.fY, fbRegler_x.fY_RE);
// Datenlogger
fbLogger(
    fSignal_1 := rE_x,
    fSignal_2 := rE_y,
    fSignal_3 := rX_x,
    fSignal_4 := rX_y,
    fSignal_5 := rW_x,
    fSignal_6 := rW_y,
    fSignal_7 := rY_R,
    fSignal_8 := rY_S,
    fSignal_9 := rY_T,
    fSignal_10 := _w7,
    nErfassung := 20000,
    bRunning := bLoggerRunning); // Logger_RET
rX_x_1 := _w5;
IF _w1 THEN _w11 := _w10 * 1; END_IF
IF _w1 THEN _w4 := _w12 * 1; END_IF
_w13 := SEL(bReAktiv, fbSignalgeno_Y_y.fY, fbRegler_y.fY_RE);
// Vorgabe im
// gesteuerten Betrieb
fbSignalgeno_Y_y(); // Signalgenerator
rY_y := _w13;
rW_y := FB_FigurePlayer_0.rW_y;
fbSignalgeno_W_y(); // Signalgenerator
// Sollwert
_w3 := rW_y - rX_y;
rE_y := _w3;
fbRegler_y(
    fE := FB_Totband_y.rPosFilt,
    eTyp := FB_ReglerParam_y.Reglertyp,
    bReset := NOT bReAktiv,
    fKr := FB_ReglerParam_y.KP,
    fTn := FB_ReglerParam_y.Ti,
    fTv := FB_ReglerParam_y.Td,
    fTvz := FB_ReglerParam_y.Tvz,
    bEnable_AWU := bAwuAktiv,
    fYlim_max := flim_max,
    fYlim_min := flim_min); // Regler
FB_ReglerParam_y(ControllerNum := ControllerNum); // FB_ReglerParam
// Regelglied
rX_x := fbFilter_X_x.fY;
rX_y := fbFilter_X_y.fY;
fbFilter_X_y(fX := MAIN.rYBallPos); // PT2
_w14 := y_r_filter.fY + rAxisOffset;
IF _w1 THEN _w16 := _w15 * 1; END_IF
xy_RST_Transformation_dynamisch_0(
    rX_X_pu := rX_x_1,
    rX_Y_pu := rX_y_1,
    rT_x := rY_x,
    rT_y := rY_y,
    rT_R_act := Main.Axis_R.DataIn.CyltronicDataInAct.ActualPosition,
    rT_S_act := Main.Axis_S.DataIn.CyltronicDataInAct.ActualPosition,
    rT_T_act := Main.Axis_T.DataIn.CyltronicDataInAct.ActualPosition); // xy_RST_Transformation_dynamisch
FB_Totband_x(rTotband := FB_ReglerParam_x.rTotband, rPos := _w9); // FB_Totband
// Zeitschritt dt
// siehe Taskhandling
RET_COMMON(fDt := GVL.rTasktime);
y_s_filter(fX := xy_RST_Transformation_dynamisch_0.rT_s, fT := ry_rst_filter); // PT1
_w17 := y_s_filter.fY + rAxisOffset;
y_r_filter(fX := xy_RST_Transformation_dynamisch_0.rT_r, fT := ry_rst_filter); // PT1
_w12 := LIMIT(rLL_rY_RST, _w18, rUL_rY_RST);
y_t_filter(fX := xy_RST_Transformation_dynamisch_0.rT_t, fT := ry_rst_filter); // PT1
_w18 := y_t_filter.fY + rAxisOffset;
_w10 := LIMIT(rLL_rY_RST, _w17, rUL_rY_RST);
_w8 := fbFilter_X_y.fY / MAIN.rMaxTouchPos;
_w15 := LIMIT(rLL_rY_RST, _w14, rUL_rY_RST);
rY_R := _w16;
rY_T := _w4;
rY_S := _w11;
MAIN.rSetPos_R := _w16;
MAIN.rSetPos_S := _w11;

END_PROGRAM

// ---- POUs/Regelungstechnik/Logger_RET.TcPOU
{attribute 'hide_all_locals' := ''}
FUNCTION_BLOCK Logger_RET
VAR_IN_OUT
	bRunning: BOOL;
END_VAR
VAR_INPUT
	fSignal_1: REAL;
	fSignal_2: REAL;
	fSignal_3: REAL;
	fSignal_4: REAL;
	fSignal_5: REAL;
	fSignal_6: REAL;
	fSignal_7: REAL;
	fSignal_8: REAL;
	fSignal_9: REAL;
	fSignal_10: REAL;
	nErfassung: UINT;
END_VAR
VAR_OUTPUT
	fActIndexProzent: REAL;
	afTime: ARRAY[0..nAnzahl] OF REAL;
	afSignal_1: ARRAY[0..nAnzahl] OF REAL;
	afSignal_2: ARRAY[0..nAnzahl] OF REAL;
	afSignal_3: ARRAY[0..nAnzahl] OF REAL;
	afSignal_4: ARRAY[0..nAnzahl] OF REAL;
	afSignal_5: ARRAY[0..nAnzahl] OF REAL;
	afSignal_6: ARRAY[0..nAnzahl] OF REAL;
	afSignal_7: ARRAY[0..nAnzahl] OF REAL;
	afSignal_8: ARRAY[0..nAnzahl] OF REAL;
	afSignal_9: ARRAY[0..nAnzahl] OF REAL;
	afSignal_10: ARRAY[0..nAnzahl] OF REAL;
END_VAR
VAR
	{attribute 'hide'}
	nStateLogger: INT := 0;
	{attribute 'hide'}
	nN: UINT;
	{attribute 'hide'}
	nIndex: UINT;
END_VAR
VAR CONSTANT
	{attribute 'hide'}
	nAnzahl: UINT := 20000;
END_VAR

// Datenlogger zur Erfassung der Sprungantwort
CASE nStateLogger OF
	0: // warte auf Sprungantwort
		fActIndexProzent := 0.0;
		nIndex := 0;
		IF bRunning THEN
			nStateLogger := 1;
		END_IF
	
	1: 	// Reset
		fActIndexProzent := 0.0;
		nIndex := 0;
		FOR nN := 0 TO nAnzahl BY 1 DO
			afTime[nN] := UINT_TO_REAL(nN)*RET_COMMON.fDt;
			afSignal_1[nN] := 0.0;
			afSignal_2[nN] := 0.0;
			afSignal_3[nN] := 0.0;
			afSignal_4[nN] := 0.0;
			afSignal_5[nN] := 0.0;
			afSignal_6[nN] := 0.0;
			afSignal_7[nN] := 0.0;
			afSignal_8[nN] := 0.0;
			afSignal_9[nN] := 0.0;
			afSignal_10[nN] := 0.0;
		END_FOR
		nStateLogger := 2;
	
	2: 
		afSignal_1[nIndex] := fSignal_1;
		afSignal_2[nIndex] := fSignal_2;
		afSignal_3[nIndex] := fSignal_3;
		afSignal_4[nIndex] := fSignal_4;
		afSignal_5[nIndex] := fSignal_5;
		afSignal_6[nIndex] := fSignal_6;
		afSignal_7[nIndex] := fSignal_7;
		afSignal_8[nIndex] := fSignal_8;
		afSignal_9[nIndex] := fSignal_9;
		afSignal_10[nIndex] := fSignal_10;
		nIndex := nIndex + 1;
		IF nIndex > MIN(nErfassung, nAnzahl) THEN
			nStateLogger := 0;
			bRunning := FALSE;
		END_IF
	
	ELSE
		nStateLogger := 0;
		bRunning := FALSE;
END_CASE
fActIndexProzent := UINT_TO_REAL(nIndex)/UINT_TO_REAL(MIN(nErfassung, nAnzahl))*100.0;

END_FUNCTION_BLOCK

// ---- POUs/Regelungstechnik/RET_COMMON.TcPOU
{attribute 'hide_all_locals' := ''}
PROGRAM RET_COMMON
VAR_INPUT
	/// Zykluszeit Main-Task
	fDt: REAL := 0.001;
END_VAR

END_PROGRAM

// ---- POUs/xy_RST_Transformation_dynamisch.TcPOU
FUNCTION_BLOCK xy_RST_Transformation_dynamisch
VAR_INPUT
	rX_X_pu: REAL;  // Aktuelle Position x-Achse (normiert auf die halbe Achslänge)
	rX_Y_pu: REAL;  // Aktuelle Position y-Achse (normiert auf die halbe Achslänge)
	rT_x: REAL; // Sollpos x-Achse
	rT_y: REAL; // Sollpos y-Achse
	rT_R_act: REAL; // Actual Position R-Axis 
	rT_S_act: REAL; // Actual Position S-Axis 
	rT_T_act: REAL; // Actual Position T-Axis 
	
END_VAR
VAR_OUTPUT
	
	rT_r: REAL; // Sollpos R-Achse
	rT_s: REAL; // Sollpos S-Achse
	rT_t: REAL; // Sollpos T-Achse	
END_VAR
VAR 
	a 		: REAL := 200; //distance to mittle of ground from Axis
	c 		: REAL := 165; //distance to middle of plate from Axis
	d		: REAL := 371; // Axis lenght when all the was in
	alpha	: REAL := 85.75; // Angle of Axis to Ground
	offset	: REAL := 34.905; // offset of axis on ground when 100mm out
	PI		: REAL := 4 * ATAN(1);
END_VAR
VAR
	r_h_R : REAL; //height of Axis plumb
	r_h_S : REAL; //height of Axis plumb
	r_h_T : REAL; //height of Axis plumb
	
	rmiddle: REAL; // hight of the middle of the plate
	rAngx : REAL; //angle for X Axis
	rAngy : REAL; //angle for Y Axis
	rKx : REAL; //
	rKy : REAL;
END_VAR

r_h_R := SQRT((d+rT_R_act)*(d+rT_R_act)-2*(d+rT_R_act)*offset*COS(alpha)+offset*offset);
r_h_S := SQRT((d+rT_S_act)*(d+rT_S_act)-2*(d+rT_S_act)*offset*COS(alpha)+offset*offset);
r_h_T := SQRT((d+rT_T_act)*(d+rT_T_act)-2*(d+rT_T_act)*offset*COS(alpha)+offset*offset);

rmiddle := (r_h_R + r_h_S + r_h_T)/3;
rAngx := RAD_TO_DEG(SIN((r_h_R - rmiddle)/c));
rAngy := RAD_TO_DEG(TAN((r_h_T - r_h_S)/285.788));
rKx := (rX_X_pu / COS(rAngx / 180 * PI));
rKy := (rX_Y_pu / COS(rAngy / 180 * PI));

rT_r := (1 - rKx) * rT_x + (0 - rKy) * rT_y;
rT_s := (-0.5 - rKx)* rT_x + ((SQRT(3) / 2) - rKy) * rT_y;
rT_t := (-0.5 - rKx)* rT_x - ((SQRT(3) / 2) + rKy) * rT_y;

END_FUNCTION_BLOCK

// ---- POUs/Regelungstechnik/PT2.TcPOU
{attribute 'hide_all_locals' := ''}
{attribute 'FBVisuCreator' := ''}
{attribute 'FBVisuCreatorPrefix' := 'RET_VISU_'}
FUNCTION_BLOCK PT2
VAR_INPUT
	{attribute 'FBVisuCreatorFormatString' := '%1.3f'}
	fX: REAL;
	{attribute 'FBVisuCreatorFormatString' := '%1.3f'}
	fK: REAL;
	{attribute 'FBVisuCreatorFormatString' := '%1.3f'}
	fT1: REAL;
	{attribute 'FBVisuCreatorFormatString' := '%1.3f'}
	fT2: REAL;
	{attribute 'FBVisuCreatorBoolColor' := 'Red'}
	bReset: BOOL;
END_VAR
VAR_OUTPUT
	{attribute 'FBVisuCreatorFormatString' := '%1.3f'}
	fY: REAL;
END_VAR
VAR
	{attribute 'hide'}
	fZeta: REAL;
	{attribute 'hide'}
	fOmega: REAL;
	{attribute 'hide'}
	fXX: REAL;
	{attribute 'hide'}
	fDx: REAL;
	{attribute 'hide'}
	fDy: REAL;
END_VAR

// Umrechnung der Faktoren in PT2s
fOmega := 1/SQRT(MAX(fT1*fT2, 0.001));
fZeta := fOmega*(fT1+fT2)/2.0;

IF bReset THEN
	reset();
END_IF

fDy := RET_COMMON.fDt*fOmega*fXX;
fDx := RET_COMMON.fDt*fOmega*(fK*fX - fY - 2*fZeta*fXX);
fXX := fXX + fDx;
fY := fY + fDy;

ACTION reset:
fXX := 0.0;
fY := 0.0;
END_ACTION

END_FUNCTION_BLOCK

// ---- POUs/Regelungstechnik/Signalgenerator.TcPOU
{attribute 'hide_all_locals' := ''}
{attribute 'FBVisuCreator' := ''}
{attribute 'FBVisuCreatorPrefix' := 'RET_VISU_'}
FUNCTION_BLOCK Signalgenerator
VAR_INPUT
	{attribute 'FBVisuCreatorFormatString' := 'd'}
	eTyp: eSignalform := eSignalform.OFF;
	{attribute 'FBVisuCreatorFormatString' := '%1.3f'}
	fOffset: REAL := 0.0;
	/// entspricht Steilheit der Rampe, d.h. 1.0 --> 1.0 dW/dt
	{attribute 'FBVisuCreatorFormatString' := '%1.3f'}
	fAmplitude: REAL := 1.0;
	{attribute 'FBVisuCreatorFormatString' := '%1.5f'}
	fFrequenz: REAL := 1.0;
	{attribute 'FBVisuCreatorFormatString' := '%1.1f'}
	fPhi: REAL := 0.0;
	{attribute 'FBVisuCreatorBoolColor' := 'Red'}
	bRauschen: BOOL;
	{attribute 'FBVisuCreatorFormatString' := '%1.3f'}
	fRauschen: REAL;
END_VAR
VAR_OUTPUT
	{attribute 'FBVisuCreatorFormatString' := '%1.3f'}
	fY: REAL;
END_VAR
VAR
	{attribute 'hide'}
	fZeit: REAL;
	{attribute 'hide'}
	fSumme: REAL;
	{attribute 'hide'}
	fbRauschen: Rauschen := (fVerstaerkung := 1.0);
	{attribute 'hide'}
	fYsin: REAL;
	{attribute 'hide'}
	fYasin: REAL;
END_VAR
VAR CONSTANT
	{attribute 'hide'}
	fPi: REAL := 3.14159265358979;
END_VAR

fZeit := fZeit + RET_COMMON.fDt;

CASE eTyp OF
	eSignalform.OFF:
		fY := 0.0;
		fSumme := 0.0;
	
	eSignalform.OFFSET:
		fY := fOffset;
		
	eSignalform.RECHTECK:
		fY := SIN(2*fPi*fFrequenz*fZeit + fPhi*fPi/180.0);
		IF fY >= 0.0 THEN
			fY := fAmplitude;
		ELSIF fY < 0.0 THEN
			fY :=  -fAmplitude;
		END_IF
		// rY := LIMIT(-100.0, rY + rOffset, 100.0);
		fY := fY + fOffset;

	eSignalform.DREIECK:
		fYsin := SIN(2*fPi*fFrequenz*fZeit + fPhi*fPi/180.0);
		fYasin := 2*ASIN(fYsin)/fPi;
		fY := fAmplitude*fYasin + fOffset;
		
	eSignalform.SINUS:
		fY := fAmplitude*SIN(2*fPi*fFrequenz*fZeit + fPhi*fPi/180.0) + fOffset;
		
	ELSE
		eTyp := eSignalform.OFF;
END_CASE
IF bRauschen AND (eTyp <> eSignalform.OFF) THEN
	fbRauschen(fVerstaerkung := fRauschen);
	fY := fY + fbRauschen.fY;
END_IF

END_FUNCTION_BLOCK

// ---- POUs/Regelungstechnik/Rauschen.TcPOU
{attribute 'hide_all_locals' := ''}
{attribute 'FBVisuCreatorPrefix' := 'RET_VISU_'}
FUNCTION_BLOCK Rauschen
VAR_INPUT
	{attribute 'FBVisuCreatorFormatString' := '%1.3f'}
	fVerstaerkung: REAL;
END_VAR
VAR_OUTPUT
	{attribute 'FBVisuCreatorFormatString' := '%1.3f'}
	fY: REAL;
END_VAR
VAR
	{attribute 'hide'}
	fSumme: REAL;
	{attribute 'hide'}
	nI: INT := 0;
END_VAR
VAR CONSTANT
	{attribute 'hide'}
